{attribute 'qualified_only'}
VAR_GLOBAL
	inputl   AT%I*   :BOOL;
	output2  AT%Q*  :BOOL;
	JoinTrack: INT;
END_VAR

(* stored: Version 1.1.0.1
   GVL GVL: Id {59c74646-7473-42d8-b33e-cdd2bd3b98de} *)
